VAR_GLOBAL
END_VAR

(* stored: Version 1.1.0.1, ProductVersion 3.1.4022.18
   GVL GVL_LAMP_GJ: Id {db708946-e289-42ed-8f83-dc3a9cd90a11} *)
